LIN {X 0,Y 59.846,Z 670.042,A -85,B 0,C 180,E1 -31316.568,E2 -31316.568} C_VEL
LIN {X 0,Y 45.695,Z 677.683,A -85,B 0,C 180,E1 -31318.66,E2 -31318.66} C_VEL
LIN {X 0,Y 31.656,Z 683.743,A -85,B 0,C 180,E1 -31322.46,E2 -31322.46} C_VEL
LIN {X 0,Y 21.304,Z 687.321,A -85,B 0,C 180,E1 -31328.233,E2 -31328.233} C_VEL
LIN {X 0,Y 8.643,Z 690.96,A -85,B 0,C 180,E1 -31355.593,E2 -31355.593} C_VEL
LIN {X 0,Y 5.756,Z 692.302,A -85,B 0,C 180,E1 -31409.996,E2 -31409.996} C_VEL
LIN {X 0,Y 8.697,Z 693.293,A -85,B 0,C 180,E1 -31463.904,E2 -31463.904} C_VEL
LIN {X 0,Y 21.327,Z 694.41,A -85,B 0,C 180,E1 -31491.333,E2 -31491.333} C_VEL
LIN {X 0,Y 28.202,Z 694.526,A -85,B 0,C 180,E1 -31495.402,E2 -31495.402} C_VEL
LIN {X 0,Y 28.134,Z 694.489,A -85,B 0,C 180,E1 -31497.714,E2 -31497.714} C_VEL
LIN {X 0,Y 17.896,Z 694.026,A -85,B 0,C 180,E1 -31505.084,E2 -31505.084} C_VEL
LIN {X 0,Y 17.896,Z 694.026,A -85,B 0,C 180,E1 -31505.084,E2 -31505.084}

QRS_NEXT_CUT()

QRS_NEXT()
QRS_HOME()

END
